PROGRAM Programma_3
VAR
    winCondition: BOOL;
	Timer: TON;
	Winner_Timer: TON;
	IN: INT;
END_VAR

// Task 3: Controleer of er een winnaar of gelijkspel is
IF GVL.game_status = 2 THEN  // Wincheck fase
    // Controleer of Speler 1 heeft gewonnen
    IF (GVL.Driehoek_1 AND GVL.Driehoek_2 AND GVL.Driehoek_3) OR
       (GVL.Driehoek_4 AND GVL.Driehoek_5 AND GVL.Driehoek_6) OR
       (GVL.Driehoek_7 AND GVL.Driehoek_8 AND GVL.Driehoek_9) OR
       (GVL.Driehoek_1 AND GVL.Driehoek_4 AND GVL.Driehoek_7) OR
       (GVL.Driehoek_2 AND GVL.Driehoek_5 AND GVL.Driehoek_8) OR
       (GVL.Driehoek_3 AND GVL.Driehoek_6 AND GVL.Driehoek_9) OR
       (GVL.Driehoek_1 AND GVL.Driehoek_5 AND GVL.Driehoek_9) OR
       (GVL.Driehoek_3 AND GVL.Driehoek_5 AND GVL.Driehoek_7) THEN
       
        // Speler 1 heeft gewonnen
        GVL.winnaar := 1;
        GVL.game_status := 3;  // Zet game status op 3 voor winnende toestand
        GVL.Player_1_Lamp_G := TRUE;  // Winnende lamp Speler 1 aan
        GVL.Player_1_Lamp := FALSE;  // Zet de lamp van Speler 1 uit
        GVL.Player_2_Lamp := FALSE;  // Zet de lamp van Speler 2 uit

    // Controleer of Speler 2 heeft gewonnen
    ELSIF (GVL.Rondje_1 AND GVL.Rondje_2 AND GVL.Rondje_3) OR
           (GVL.Rondje_4 AND GVL.Rondje_5 AND GVL.Rondje_6) OR
           (GVL.Rondje_7 AND GVL.Rondje_8 AND GVL.Rondje_9) OR
           (GVL.Rondje_1 AND GVL.Rondje_4 AND GVL.Rondje_7) OR
           (GVL.Rondje_2 AND GVL.Rondje_5 AND GVL.Rondje_8) OR
           (GVL.Rondje_3 AND GVL.Rondje_6 AND GVL.Rondje_9) OR
           (GVL.Rondje_1 AND GVL.Rondje_5 AND GVL.Rondje_9) OR
           (GVL.Rondje_3 AND GVL.Rondje_5 AND GVL.Rondje_7) THEN

        // Speler 2 heeft gewonnen
        GVL.winnaar := 2;
        GVL.game_status := 3;  // Zet game status op 3 voor winnende toestand
        GVL.Player_2_Lamp_G := TRUE;  // Winnende lamp Speler 2 aan
        GVL.Player_1_Lamp := FALSE;  // Zet de lamp van Speler 1 uit
        GVL.Player_2_Lamp := FALSE;  // Zet de lamp van Speler 2 uit

    ELSE
        // Als er geen winnaar is, controleer dan of het gelijkspel is
        IF (GVL.Driehoek_1 OR GVL.Rondje_1) AND
           (GVL.Driehoek_2 OR GVL.Rondje_2) AND
           (GVL.Driehoek_3 OR GVL.Rondje_3) AND
           (GVL.Driehoek_4 OR GVL.Rondje_4) AND
           (GVL.Driehoek_5 OR GVL.Rondje_5) AND
           (GVL.Driehoek_6 OR GVL.Rondje_6) AND
           (GVL.Driehoek_7 OR GVL.Rondje_7) AND
           (GVL.Driehoek_8 OR GVL.Rondje_8) AND
           (GVL.Driehoek_9 OR GVL.Rondje_9) THEN
            // Het is gelijkspel
            GVL.Gelijkspel := TRUE;  // Zet status naar gelijkspel
		    GVL.Player_1_Lamp := FALSE;  // Zet de lamp van Speler 1 uit na wachttijd
			GVL.Player_2_Lamp := FALSE;
        ELSE
            // Er zijn nog lege vakken, geen gelijkspel
            GVL.game_status := 1;  // Ga terug naar de beurtfase
        END_IF
    END_IF
END_IF

END_PROGRAM

(* stored: Version 1.1.0.1, ProductVersion 3.1.4024.12
   POU Programma_3: Id {70a6b97a-964e-4e36-9a7b-67e0026594f5}, SpecialFunc None *)
